(* PLC project KinIn_v3.project, CODESYS CODESYS V3.5 SP19 *)
(* stored: creationDateTime 2025-01-20T16:27:50.975359, modificationDateTime 2025-01-20T16:17:39.6822999 *)

FUNCTION_BLOCK transpose
  VAR
    t_count1_i : DINT;  (* ------------- *)
    t_count1_j : DINT;
  END_VAR
  VAR_INPUT
    {attribute 'variable_length_array_original_scope' := 'Inout'}
    {attribute 'variable_length_array' := 'ARRAY[*,*] OF REAL'}
    {attribute 'Dimensions' := '2'}
    B : POINTER TO REAL;
    {attribute 'variable_length_array_original_scope' := 'Inout'}
    {attribute 'variable_length_array' := 'ARRAY[*,*] OF REAL'}
    {attribute 'Dimensions' := '2'}
    Bt : POINTER TO REAL;
  END_VAR

            
//----creating the code for the transpose--------
FOR t_count1_i:=LOWER_BOUND(B,1) TO UPPER_BOUND(B,1) DO
	FOR t_count1_j:=LOWER_BOUND(B,2) TO UPPER_BOUND(B,2) DO
		Bt[t_count1_j,t_count1_i]:=B[t_count1_i,t_count1_j];//transpose the indexes
	END_FOR
	
END_FOR
          
END_FUNCTION_BLOCK
